{attribute 'linkalways'} 
{attribute 'no_explicit_call' := 'This FB is a CLASS and must be accessed using methods or properties'}
{attribute 'enable_dynamic_creation'}
FUNCTION_BLOCK Node_ContainerType_Vector_TcVnVector2_INT EXTENDS Node
VAR
    out : _GUID;
END_VAR

METHOD PUBLIC  Clone : I_Node
VAR
	pNode : POINTER TO Node_ContainerType_Vector_TcVnVector2_INT;
END_VAR
pNode := __NEW(Node_ContainerType_Vector_TcVnVector2_INT);
Clone := pNode^;
END_METHOD

METHOD FB_init : BOOL
VAR_INPUT
	bInitRetains : BOOL; // if TRUE, the retain variables are initialized (warm start / cold start)
	bInCopyCode : BOOL;  // if TRUE, the instance afterwards gets moved into the copy code (online change)
END_VAR
AddOutput('out', out);
END_METHOD

METHOD PROTECTED OnExecute
out.Value := ContainerType_Vector_TcVnVector2_INT;
END_METHOD

END_FUNCTION_BLOCK

(* stored: Version 1.1.0.1, ProductVersion 3.1.4026.17
   POU Node_ContainerType_Vector_TcVnVector2_INT: Id {401df609-453f-002e-2740-b3000b8643bf}, SpecialFunc None
   Folder Constructor: Id {3efbc0a8-0277-05a2-3ff3-229a08f28d2f}
   Method Clone: Id {5683c3b4-75a0-0ba9-222b-8cdd6ae09838}
   Method FB_init: Id {8044ec53-ff3e-070d-3a01-e0d00e01acda}
   Method OnExecute: Id {c03caa3e-2adb-011c-1178-f4ad7e0b8533} *)
